(* Logix 5000 project; controller AMANA_DC_PLANT_01 vendor 1 type 14 code 164 rev 31.12; software revision 31.02; part 4 of 9 *)
(* tags used below, declared in another part *)
   Break_1stStation : BOOL;
   Break_LineWide : BOOL;
   Break_WorkCenter : BOOL;
   Break_Workstation : BOOL;
   Local_Timer : TIMER[10];
   LN00_1st_Station_Break_Code : DINT;
   LN00_FPY : REAL;
   LN00_MLC_Downtime : BOOL;
   LN00_Schedule : UDT_Current_Status;
   LN00_SNModel_MSG : MESSAGE;
   LN00_to_DC1_Main_Messages_0 : DINT[40];
   LN00_to_DC1_Main_Messages_1 : DINT[120];
   LN00_to_DC1_Main_Messages_2 : DINT[120];
   LN00_to_DC1_Main_Messages_3 : DINT[120];
   LN00_to_DC1_Main_Messages_4 : DINT[120];
   LN00_to_DC1_Main_Messages_5 : DINT[120];
   LN00_to_DC1_Main_MSG1 : MESSAGE;
   LN00_to_DC1_Main_MSG2 : MESSAGE;
   LN00_to_DC1_Main_MSG3 : MESSAGE;
   LN00_to_DC1_Main_MSG4 : MESSAGE;
   LN00_to_DC1_Main_MSG5 : MESSAGE;
   LN00_to_DC1_Main_MSG6 : MESSAGE;
   LN00DAM01 : DINT;
   LN00DAM02 : DINT;
   LN00DAM03 : DINT;
   LN00DAM04 : DINT;
   LN00DAM05 : DINT;
   LN00DAM06 : DINT;
   LN00DAM07 : DINT;
   LN00DAM08 : DINT;
   LN00DAM09 : DINT;
   LN00DBM02 : DINT;
   LN00DBM03 : DINT;
   LN00DCM04 : DINT;
   LN00DCM05 : DINT;
   LN00DCM06 : DINT;
   LN00DCM07 : DINT;
   LN00DCM08 : DINT;
   LN00DCM09 : DINT;
   LN00DCM10 : DINT;
   LN00DCM11 : DINT;
   LN00DCM12 : DINT;
   LN00DCM13 : DINT;
   LN00DCM14 : DINT;
   LN00DCM15 : DINT;
   LN00DCM16 : DINT;
   LN00DCM17 : DINT;
   LN00DCM18 : DINT;
   LN00DCM19 : DINT;
   LN00DCM20 : DINT;
   LN00DCM21 : DINT;
   LN00DCM22 : DINT;
   LN00DCM23 : DINT;
   LN00DCM24 : DINT;
   LN00DCM25 : DINT;
   LN00DCM26 : DINT;
   LN00DCM27 : DINT;
   LN00DCM28 : DINT;
   LN00DCM29 : DINT;
   LN00DCM30 : DINT;
   LN00DCM31 : DINT;
   LN00DCM32 : DINT;
   LN00DCM33 : DINT;
   LN00DCM34 : DINT;
   LN00DCM35 : DINT;
   LN00DCM36 : DINT;
   LN00DCM37 : DINT;
   LN00DCM38 : DINT;
   LN00DCM39 : DINT;
   LN00DCM40 : DINT;
   LN00DDM01 : DINT;
   LN00DDM02 : DINT;
   LN00DDM03 : DINT;
   LN00DDM04 : DINT;
   LN00DDM05 : DINT;
   LN00DDM06 : DINT;
   LN00DDM07 : DINT;
   LN00DDM08 : DINT;
   LN00DDM09 : DINT;
   LN00DDM10 : DINT;
   LN00DDM11 : DINT;
   LN00DDM12 : DINT;
   LN00DDM13 : DINT;
   LN00DDM14 : DINT;
   LN00DDM15 : DINT;
   LN00DDM16 : DINT;
   LN00DDM17 : DINT;
   LN00DDM18 : DINT;
   LN00DDM19 : DINT;
   LN00DDM20 : DINT;
   LN00DDM21 : DINT;
   LN00DDM22 : DINT;
   LN00DDM23 : DINT;
   LN00DDM24 : DINT;
   LN00DDM25 : DINT;
   LN00DDM26 : DINT;
   LN00DDM27 : DINT;
   LN00DDM28 : DINT;
   LN00DEM01 : DINT;
   LN00DEM02 : DINT;
   LN00DEM03 : DINT;
   LN00DEM04 : DINT;
   LN00DEM05 : DINT;
   LN00EAM00 : DINT;
   LN00EBM00 : DINT;
   LN00EDM00 : DINT;
(* LN00, continued *)

ROUTINE R03_DataFromLines   (* ladder *)
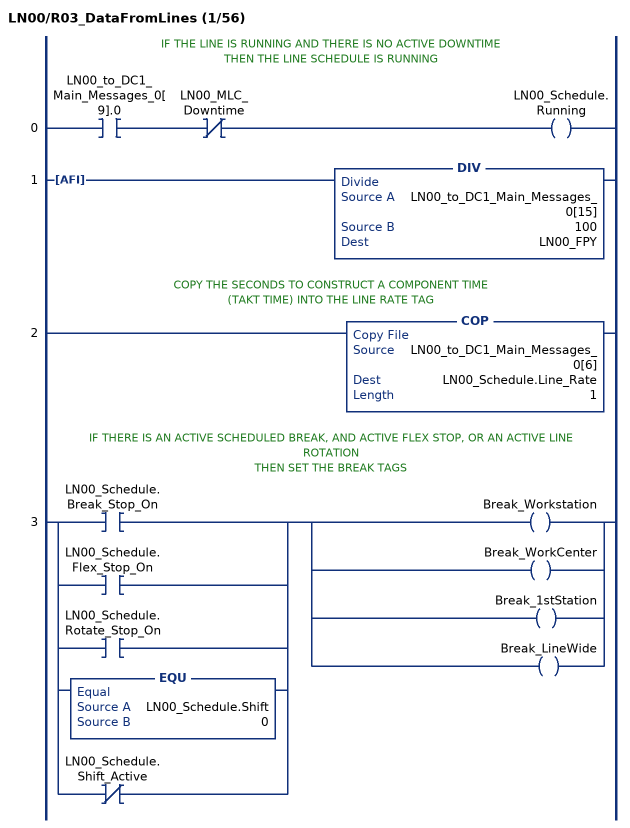
   // IF THE LINE IS RUNNING AND THERE IS NO ACTIVE DOWNTIME
   // THEN THE LINE SCHEDULE IS RUNNING
   0: XIC(LN00_to_DC1_Main_Messages_0[9].0)XIO(LN00_MLC_Downtime)OTE(LN00_Schedule.Running);
   1: AFI()DIV(LN00_to_DC1_Main_Messages_0[15],100,LN00_FPY);
   // COPY THE SECONDS TO CONSTRUCT A COMPONENT TIME
   // (TAKT TIME) INTO THE LINE RATE TAG
   2: COP(LN00_to_DC1_Main_Messages_0[6],LN00_Schedule.Line_Rate,1);
   // IF THERE IS AN ACTIVE SCHEDULED BREAK, AND ACTIVE FLEX STOP, OR AN ACTIVE LINE ROTATION
   // THEN SET THE BREAK TAGS
   3: [XIC(LN00_Schedule.Break_Stop_On) ,XIC(LN00_Schedule.Flex_Stop_On) ,XIC(LN00_Schedule.Rotate_Stop_On) ,EQU(LN00_Schedule.Shift,0) ,XIO(LN00_Schedule.Shift_Active) ][OTE(Break_Workstation) ,OTE(Break_WorkCenter) ,OTE(Break_1stStation) ,OTE(Break_LineWide) ];
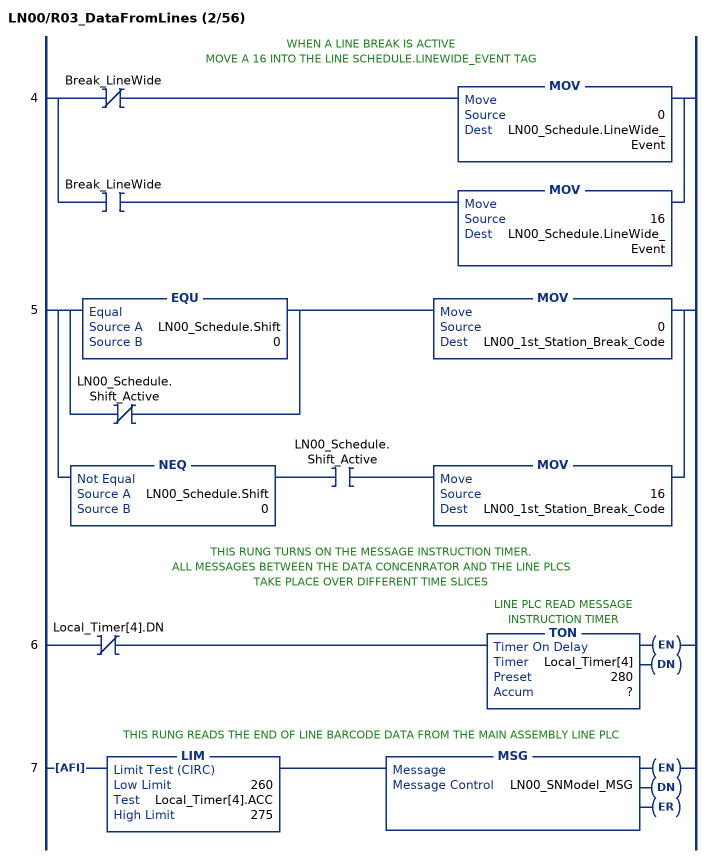
   // WHEN A LINE BREAK IS ACTIVE
   // MOVE A 16 INTO THE LINE SCHEDULE.LINEWIDE_EVENT TAG
   4: [XIO(Break_LineWide) MOV(0,LN00_Schedule.LineWide_Event) ,XIC(Break_LineWide) MOV(16,LN00_Schedule.LineWide_Event) ];
   5: [[EQU(LN00_Schedule.Shift,0) ,XIO(LN00_Schedule.Shift_Active) ] MOV(0,LN00_1st_Station_Break_Code) ,NEQ(LN00_Schedule.Shift,0) XIC(LN00_Schedule.Shift_Active) MOV(16,LN00_1st_Station_Break_Code) ];
   // THIS RUNG TURNS ON THE MESSAGE INSTRUCTION TIMER.
   // ALL MESSAGES BETWEEN THE DATA CONCENRATOR AND THE LINE PLCS
   // TAKE PLACE OVER DIFFERENT TIME SLICES
   6: XIO(Local_Timer[4].DN)TON(Local_Timer[4],?,?);
   // THIS RUNG READS THE END OF LINE BARCODE DATA FROM THE MAIN ASSEMBLY LINE PLC
   7: AFI()LIM(260,Local_Timer[4].ACC,275)MSG(LN00_SNModel_MSG);
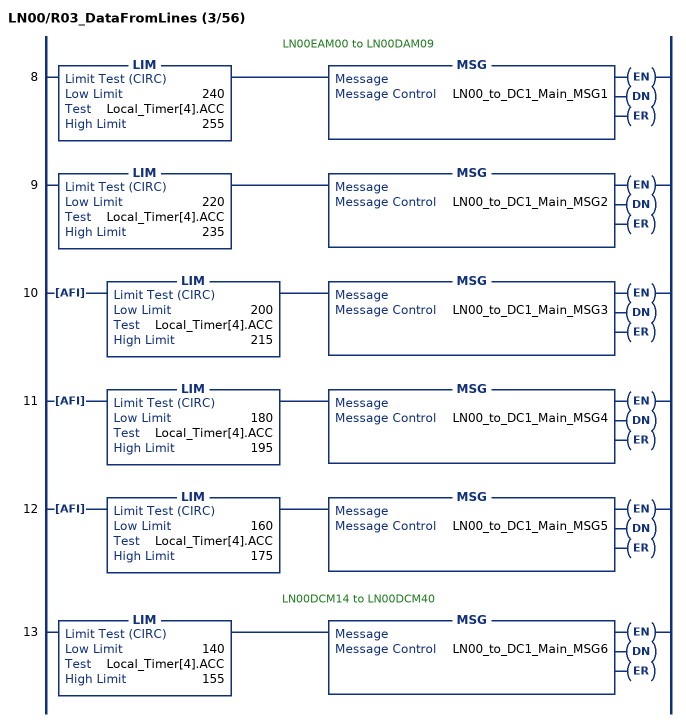
   // LN00EAM00 to LN00DAM09
   8: LIM(240,Local_Timer[4].ACC,255)MSG(LN00_to_DC1_Main_MSG1);
   9: LIM(220,Local_Timer[4].ACC,235)MSG(LN00_to_DC1_Main_MSG2);
   10: AFI()LIM(200,Local_Timer[4].ACC,215)MSG(LN00_to_DC1_Main_MSG3);
   11: AFI()LIM(180,Local_Timer[4].ACC,195)MSG(LN00_to_DC1_Main_MSG4);
   12: AFI()LIM(160,Local_Timer[4].ACC,175)MSG(LN00_to_DC1_Main_MSG5);
   // LN00DCM14 to LN00DCM40
   13: LIM(140,Local_Timer[4].ACC,155)MSG(LN00_to_DC1_Main_MSG6);
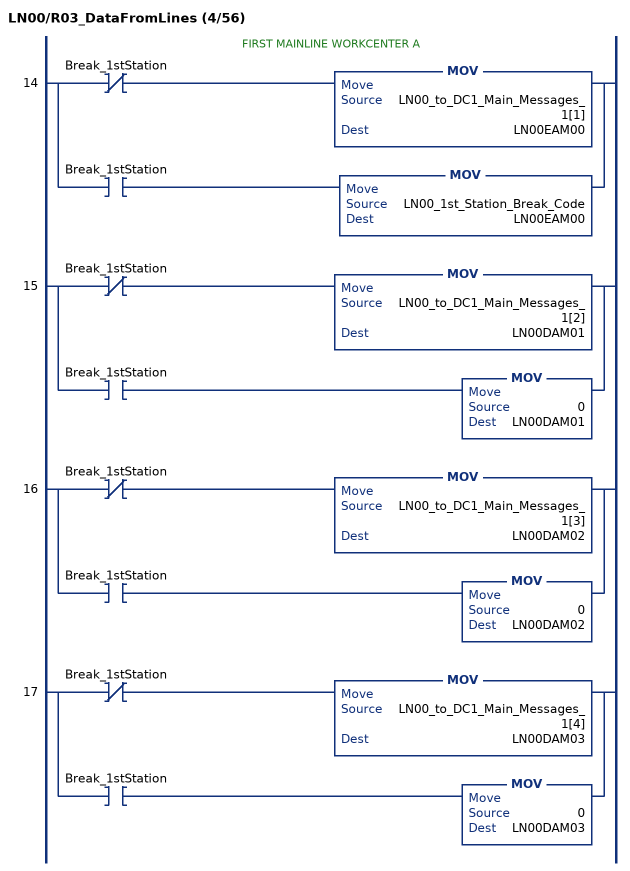
   // FIRST MAINLINE WORKCENTER A
   14: [XIO(Break_1stStation) MOV(LN00_to_DC1_Main_Messages_1[1],LN00EAM00) ,XIC(Break_1stStation) MOV(LN00_1st_Station_Break_Code,LN00EAM00) ];
   15: [XIO(Break_1stStation) MOV(LN00_to_DC1_Main_Messages_1[2],LN00DAM01) ,XIC(Break_1stStation) MOV(0,LN00DAM01) ];
   16: [XIO(Break_1stStation) MOV(LN00_to_DC1_Main_Messages_1[3],LN00DAM02) ,XIC(Break_1stStation) MOV(0,LN00DAM02) ];
   17: [XIO(Break_1stStation) MOV(LN00_to_DC1_Main_Messages_1[4],LN00DAM03) ,XIC(Break_1stStation) MOV(0,LN00DAM03) ];
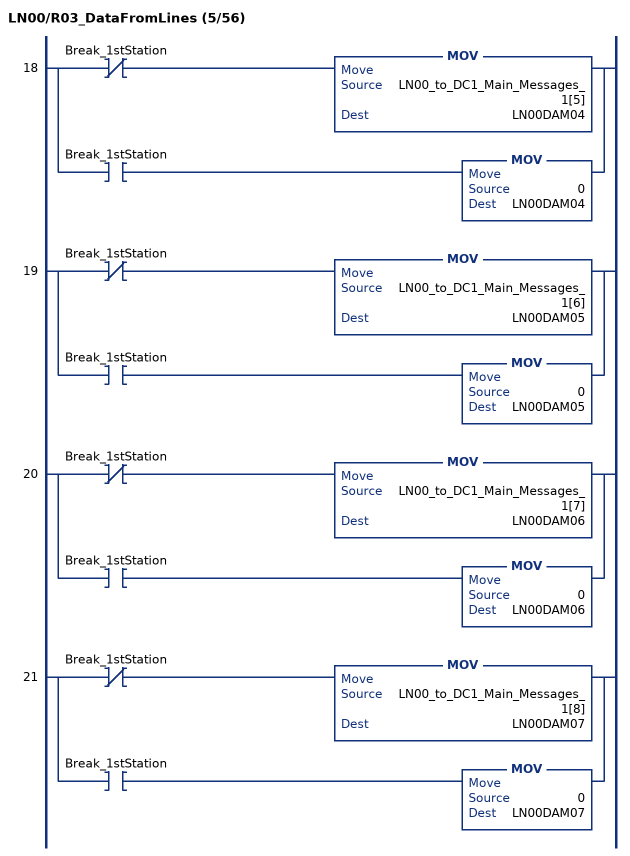
   18: [XIO(Break_1stStation) MOV(LN00_to_DC1_Main_Messages_1[5],LN00DAM04) ,XIC(Break_1stStation) MOV(0,LN00DAM04) ];
   19: [XIO(Break_1stStation) MOV(LN00_to_DC1_Main_Messages_1[6],LN00DAM05) ,XIC(Break_1stStation) MOV(0,LN00DAM05) ];
   20: [XIO(Break_1stStation) MOV(LN00_to_DC1_Main_Messages_1[7],LN00DAM06) ,XIC(Break_1stStation) MOV(0,LN00DAM06) ];
   21: [XIO(Break_1stStation) MOV(LN00_to_DC1_Main_Messages_1[8],LN00DAM07) ,XIC(Break_1stStation) MOV(0,LN00DAM07) ];
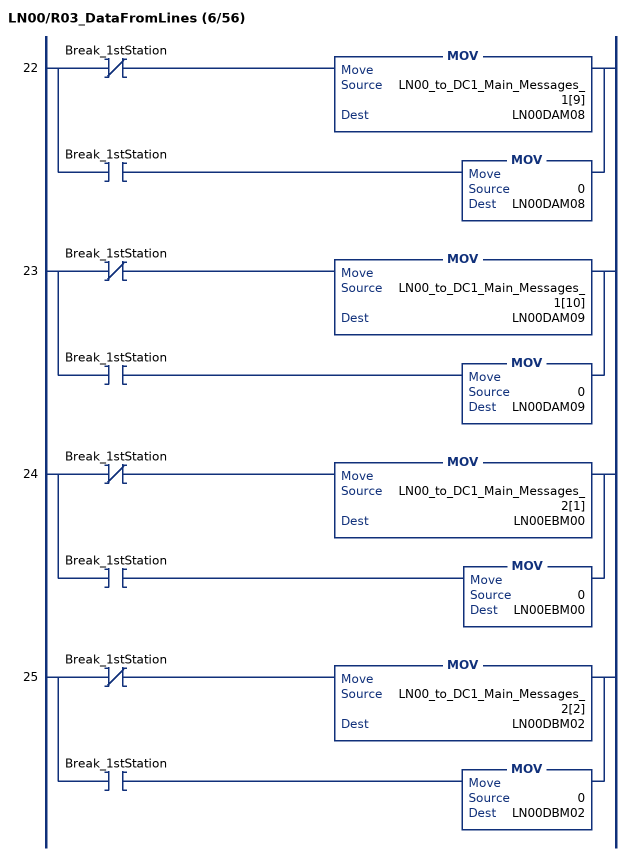
   22: [XIO(Break_1stStation) MOV(LN00_to_DC1_Main_Messages_1[9],LN00DAM08) ,XIC(Break_1stStation) MOV(0,LN00DAM08) ];
   23: [XIO(Break_1stStation) MOV(LN00_to_DC1_Main_Messages_1[10],LN00DAM09) ,XIC(Break_1stStation) MOV(0,LN00DAM09) ];
   24: [XIO(Break_1stStation) MOV(LN00_to_DC1_Main_Messages_2[1],LN00EBM00) ,XIC(Break_1stStation) MOV(0,LN00EBM00) ];
   25: [XIO(Break_1stStation) MOV(LN00_to_DC1_Main_Messages_2[2],LN00DBM02) ,XIC(Break_1stStation) MOV(0,LN00DBM02) ];
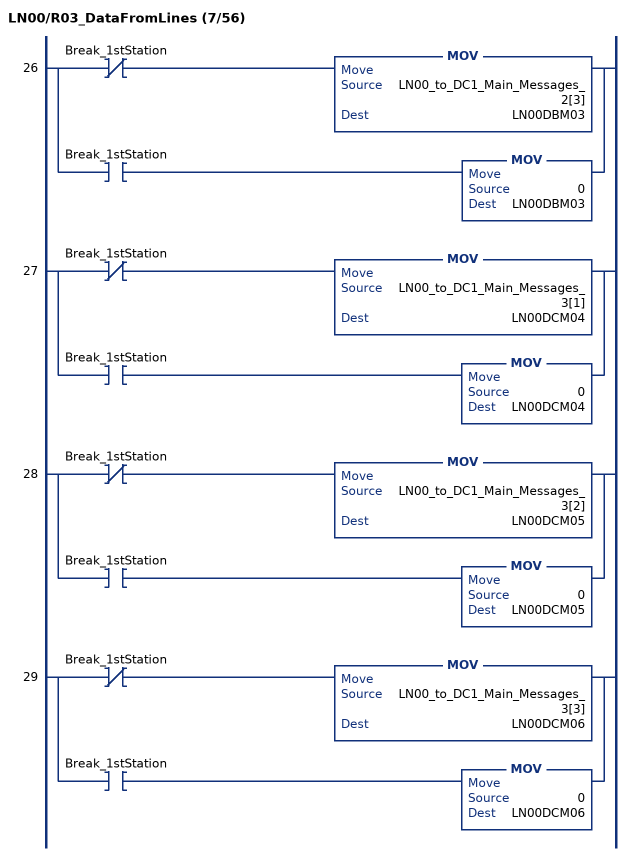
   26: [XIO(Break_1stStation) MOV(LN00_to_DC1_Main_Messages_2[3],LN00DBM03) ,XIC(Break_1stStation) MOV(0,LN00DBM03) ];
   27: [XIO(Break_1stStation) MOV(LN00_to_DC1_Main_Messages_3[1],LN00DCM04) ,XIC(Break_1stStation) MOV(0,LN00DCM04) ];
   28: [XIO(Break_1stStation) MOV(LN00_to_DC1_Main_Messages_3[2],LN00DCM05) ,XIC(Break_1stStation) MOV(0,LN00DCM05) ];
   29: [XIO(Break_1stStation) MOV(LN00_to_DC1_Main_Messages_3[3],LN00DCM06) ,XIC(Break_1stStation) MOV(0,LN00DCM06) ];
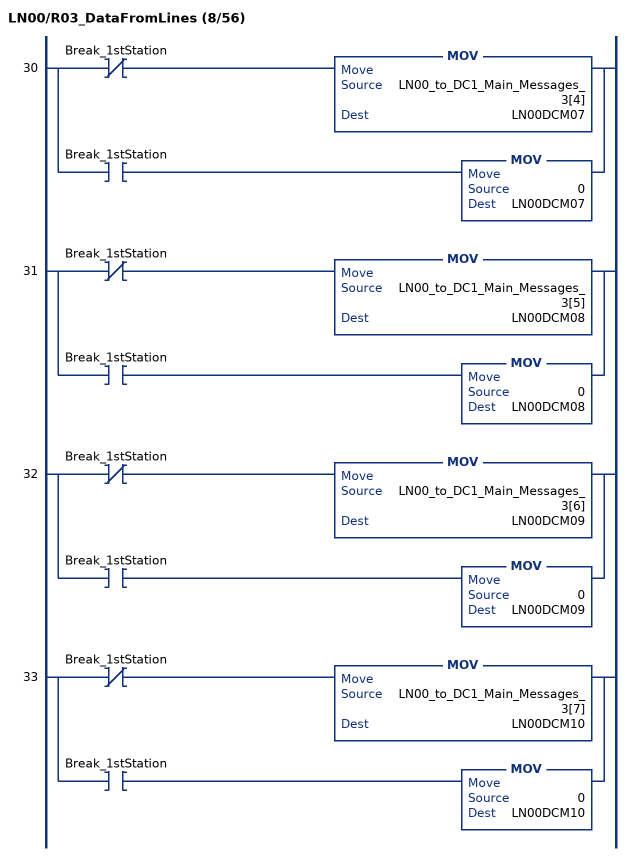
   30: [XIO(Break_1stStation) MOV(LN00_to_DC1_Main_Messages_3[4],LN00DCM07) ,XIC(Break_1stStation) MOV(0,LN00DCM07) ];
   31: [XIO(Break_1stStation) MOV(LN00_to_DC1_Main_Messages_3[5],LN00DCM08) ,XIC(Break_1stStation) MOV(0,LN00DCM08) ];
   32: [XIO(Break_1stStation) MOV(LN00_to_DC1_Main_Messages_3[6],LN00DCM09) ,XIC(Break_1stStation) MOV(0,LN00DCM09) ];
   33: [XIO(Break_1stStation) MOV(LN00_to_DC1_Main_Messages_3[7],LN00DCM10) ,XIC(Break_1stStation) MOV(0,LN00DCM10) ];
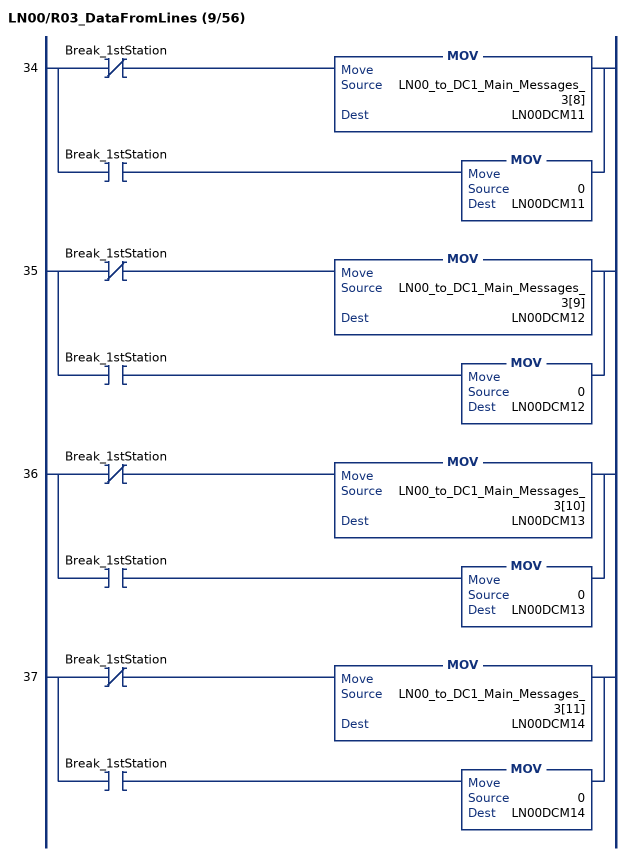
   34: [XIO(Break_1stStation) MOV(LN00_to_DC1_Main_Messages_3[8],LN00DCM11) ,XIC(Break_1stStation) MOV(0,LN00DCM11) ];
   35: [XIO(Break_1stStation) MOV(LN00_to_DC1_Main_Messages_3[9],LN00DCM12) ,XIC(Break_1stStation) MOV(0,LN00DCM12) ];
   36: [XIO(Break_1stStation) MOV(LN00_to_DC1_Main_Messages_3[10],LN00DCM13) ,XIC(Break_1stStation) MOV(0,LN00DCM13) ];
   37: [XIO(Break_1stStation) MOV(LN00_to_DC1_Main_Messages_3[11],LN00DCM14) ,XIC(Break_1stStation) MOV(0,LN00DCM14) ];
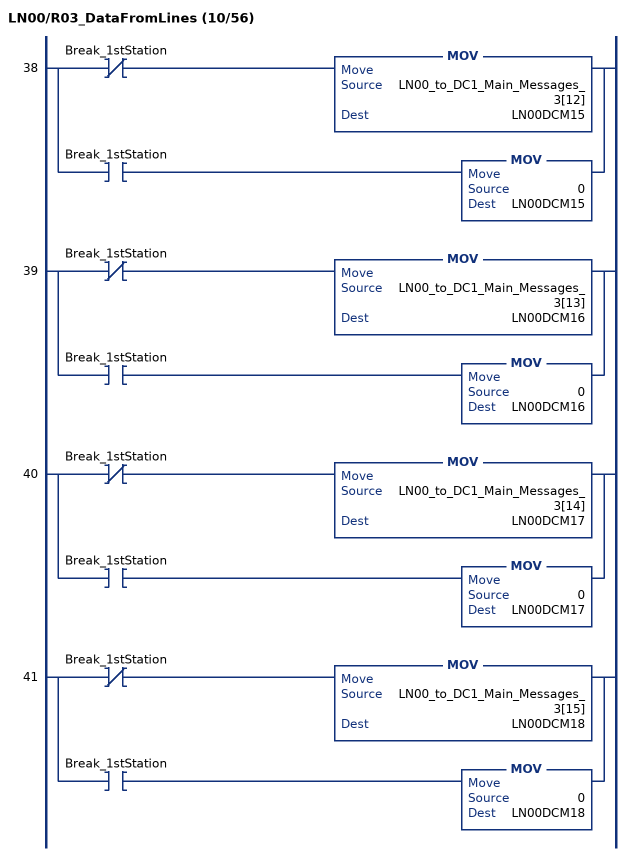
   38: [XIO(Break_1stStation) MOV(LN00_to_DC1_Main_Messages_3[12],LN00DCM15) ,XIC(Break_1stStation) MOV(0,LN00DCM15) ];
   39: [XIO(Break_1stStation) MOV(LN00_to_DC1_Main_Messages_3[13],LN00DCM16) ,XIC(Break_1stStation) MOV(0,LN00DCM16) ];
   40: [XIO(Break_1stStation) MOV(LN00_to_DC1_Main_Messages_3[14],LN00DCM17) ,XIC(Break_1stStation) MOV(0,LN00DCM17) ];
   41: [XIO(Break_1stStation) MOV(LN00_to_DC1_Main_Messages_3[15],LN00DCM18) ,XIC(Break_1stStation) MOV(0,LN00DCM18) ];
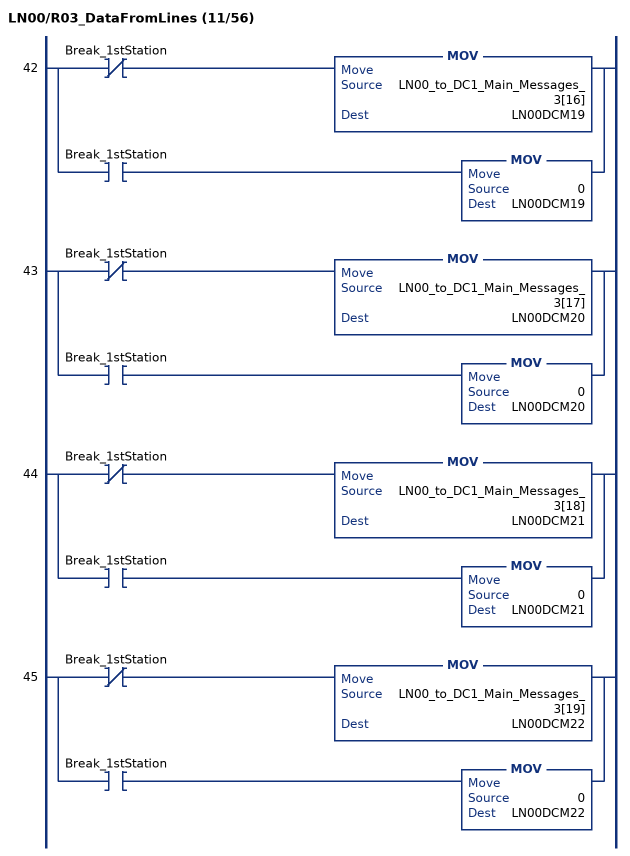
   42: [XIO(Break_1stStation) MOV(LN00_to_DC1_Main_Messages_3[16],LN00DCM19) ,XIC(Break_1stStation) MOV(0,LN00DCM19) ];
   43: [XIO(Break_1stStation) MOV(LN00_to_DC1_Main_Messages_3[17],LN00DCM20) ,XIC(Break_1stStation) MOV(0,LN00DCM20) ];
   44: [XIO(Break_1stStation) MOV(LN00_to_DC1_Main_Messages_3[18],LN00DCM21) ,XIC(Break_1stStation) MOV(0,LN00DCM21) ];
   45: [XIO(Break_1stStation) MOV(LN00_to_DC1_Main_Messages_3[19],LN00DCM22) ,XIC(Break_1stStation) MOV(0,LN00DCM22) ];
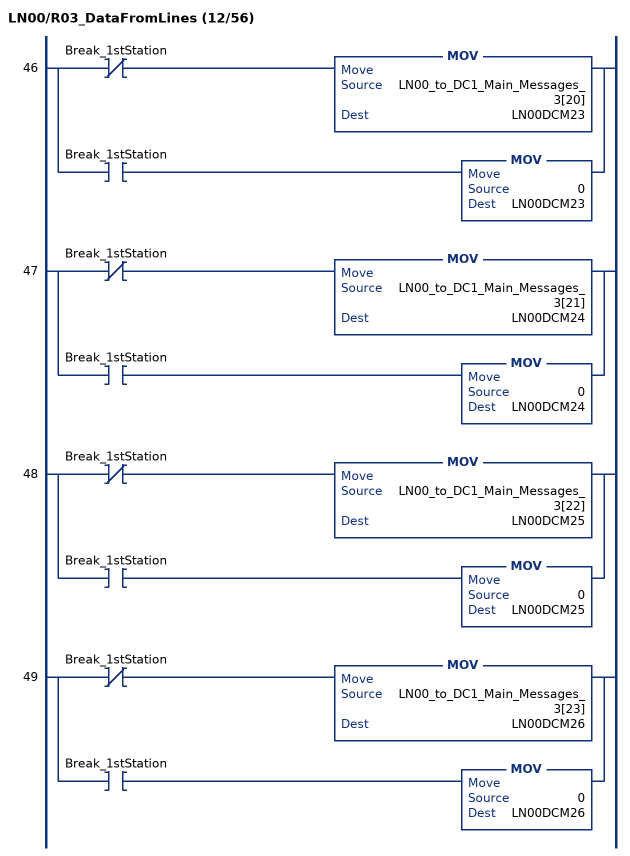
   46: [XIO(Break_1stStation) MOV(LN00_to_DC1_Main_Messages_3[20],LN00DCM23) ,XIC(Break_1stStation) MOV(0,LN00DCM23) ];
   47: [XIO(Break_1stStation) MOV(LN00_to_DC1_Main_Messages_3[21],LN00DCM24) ,XIC(Break_1stStation) MOV(0,LN00DCM24) ];
   48: [XIO(Break_1stStation) MOV(LN00_to_DC1_Main_Messages_3[22],LN00DCM25) ,XIC(Break_1stStation) MOV(0,LN00DCM25) ];
   49: [XIO(Break_1stStation) MOV(LN00_to_DC1_Main_Messages_3[23],LN00DCM26) ,XIC(Break_1stStation) MOV(0,LN00DCM26) ];
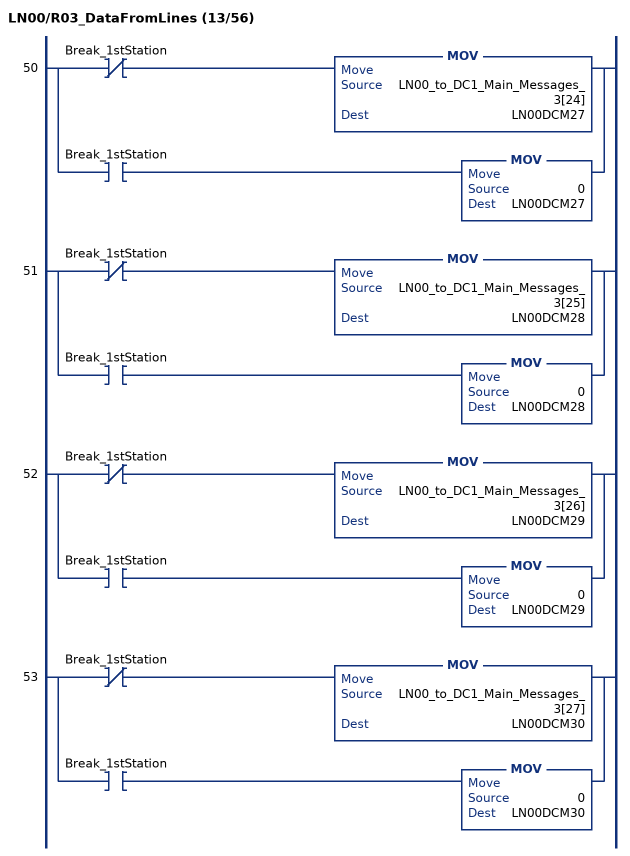
   50: [XIO(Break_1stStation) MOV(LN00_to_DC1_Main_Messages_3[24],LN00DCM27) ,XIC(Break_1stStation) MOV(0,LN00DCM27) ];
   51: [XIO(Break_1stStation) MOV(LN00_to_DC1_Main_Messages_3[25],LN00DCM28) ,XIC(Break_1stStation) MOV(0,LN00DCM28) ];
   52: [XIO(Break_1stStation) MOV(LN00_to_DC1_Main_Messages_3[26],LN00DCM29) ,XIC(Break_1stStation) MOV(0,LN00DCM29) ];
   53: [XIO(Break_1stStation) MOV(LN00_to_DC1_Main_Messages_3[27],LN00DCM30) ,XIC(Break_1stStation) MOV(0,LN00DCM30) ];
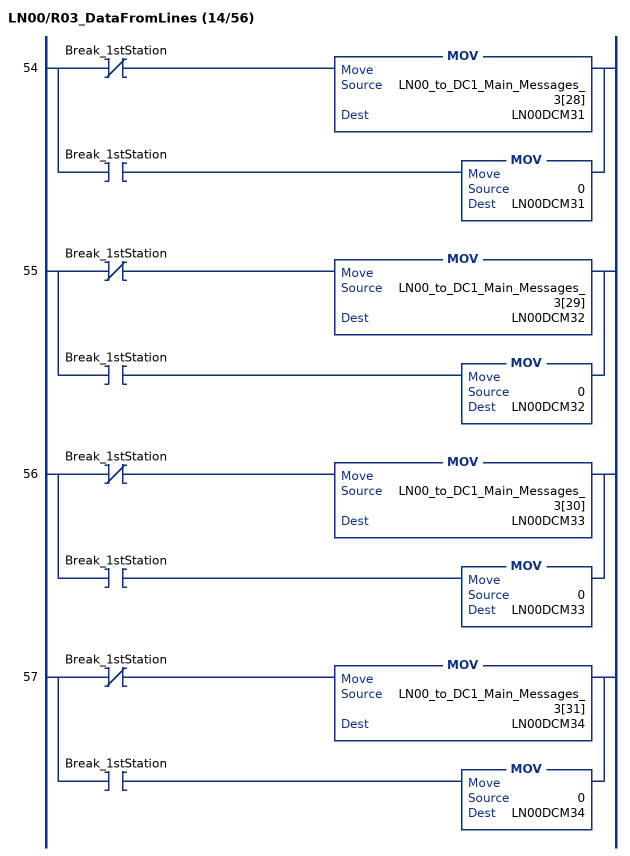
   54: [XIO(Break_1stStation) MOV(LN00_to_DC1_Main_Messages_3[28],LN00DCM31) ,XIC(Break_1stStation) MOV(0,LN00DCM31) ];
   55: [XIO(Break_1stStation) MOV(LN00_to_DC1_Main_Messages_3[29],LN00DCM32) ,XIC(Break_1stStation) MOV(0,LN00DCM32) ];
   56: [XIO(Break_1stStation) MOV(LN00_to_DC1_Main_Messages_3[30],LN00DCM33) ,XIC(Break_1stStation) MOV(0,LN00DCM33) ];
   57: [XIO(Break_1stStation) MOV(LN00_to_DC1_Main_Messages_3[31],LN00DCM34) ,XIC(Break_1stStation) MOV(0,LN00DCM34) ];
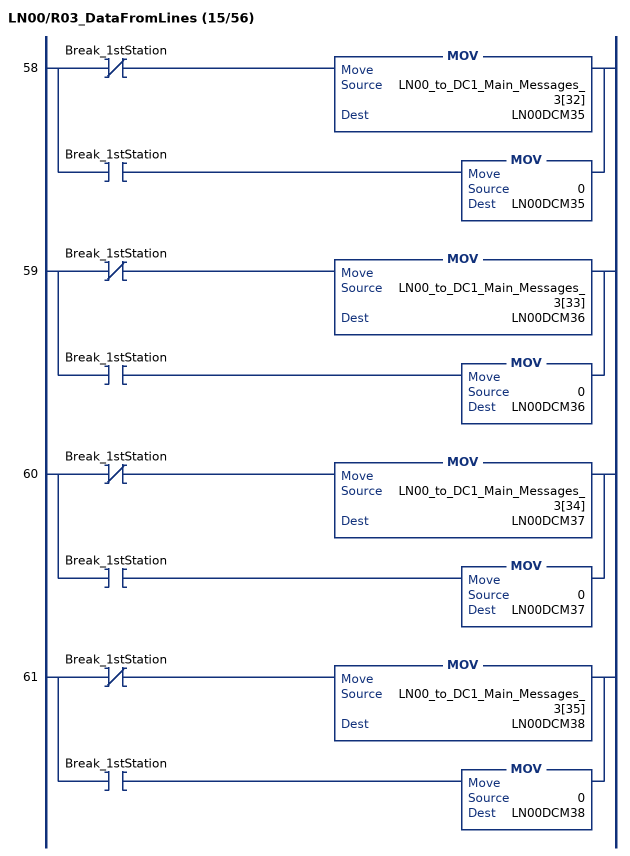
   58: [XIO(Break_1stStation) MOV(LN00_to_DC1_Main_Messages_3[32],LN00DCM35) ,XIC(Break_1stStation) MOV(0,LN00DCM35) ];
   59: [XIO(Break_1stStation) MOV(LN00_to_DC1_Main_Messages_3[33],LN00DCM36) ,XIC(Break_1stStation) MOV(0,LN00DCM36) ];
   60: [XIO(Break_1stStation) MOV(LN00_to_DC1_Main_Messages_3[34],LN00DCM37) ,XIC(Break_1stStation) MOV(0,LN00DCM37) ];
   61: [XIO(Break_1stStation) MOV(LN00_to_DC1_Main_Messages_3[35],LN00DCM38) ,XIC(Break_1stStation) MOV(0,LN00DCM38) ];
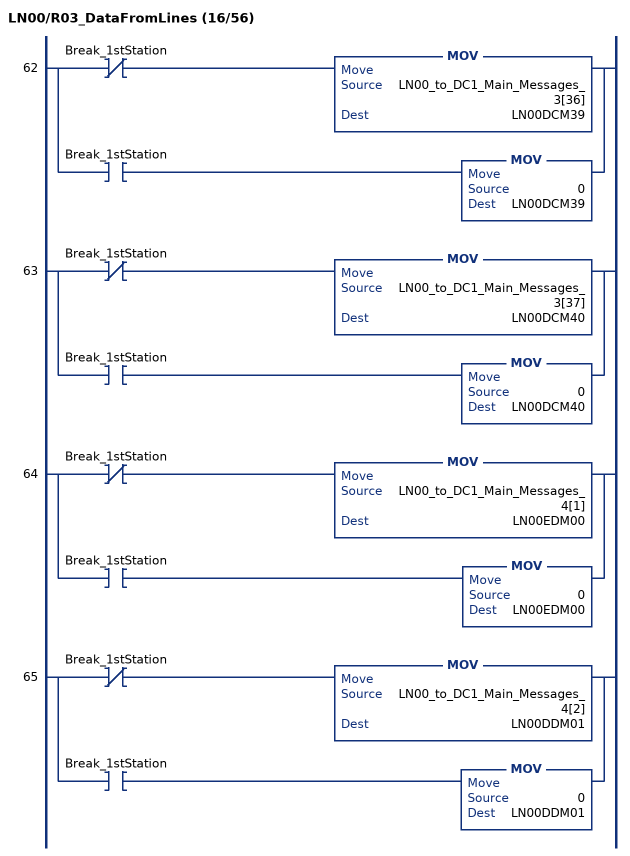
   62: [XIO(Break_1stStation) MOV(LN00_to_DC1_Main_Messages_3[36],LN00DCM39) ,XIC(Break_1stStation) MOV(0,LN00DCM39) ];
   63: [XIO(Break_1stStation) MOV(LN00_to_DC1_Main_Messages_3[37],LN00DCM40) ,XIC(Break_1stStation) MOV(0,LN00DCM40) ];
   64: [XIO(Break_1stStation) MOV(LN00_to_DC1_Main_Messages_4[1],LN00EDM00) ,XIC(Break_1stStation) MOV(0,LN00EDM00) ];
   65: [XIO(Break_1stStation) MOV(LN00_to_DC1_Main_Messages_4[2],LN00DDM01) ,XIC(Break_1stStation) MOV(0,LN00DDM01) ];
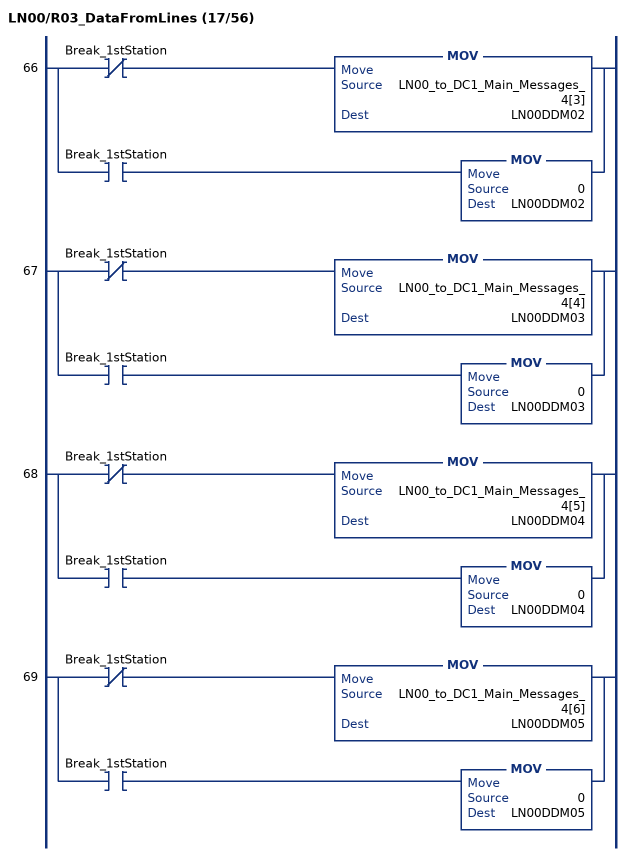
   66: [XIO(Break_1stStation) MOV(LN00_to_DC1_Main_Messages_4[3],LN00DDM02) ,XIC(Break_1stStation) MOV(0,LN00DDM02) ];
   67: [XIO(Break_1stStation) MOV(LN00_to_DC1_Main_Messages_4[4],LN00DDM03) ,XIC(Break_1stStation) MOV(0,LN00DDM03) ];
   68: [XIO(Break_1stStation) MOV(LN00_to_DC1_Main_Messages_4[5],LN00DDM04) ,XIC(Break_1stStation) MOV(0,LN00DDM04) ];
   69: [XIO(Break_1stStation) MOV(LN00_to_DC1_Main_Messages_4[6],LN00DDM05) ,XIC(Break_1stStation) MOV(0,LN00DDM05) ];
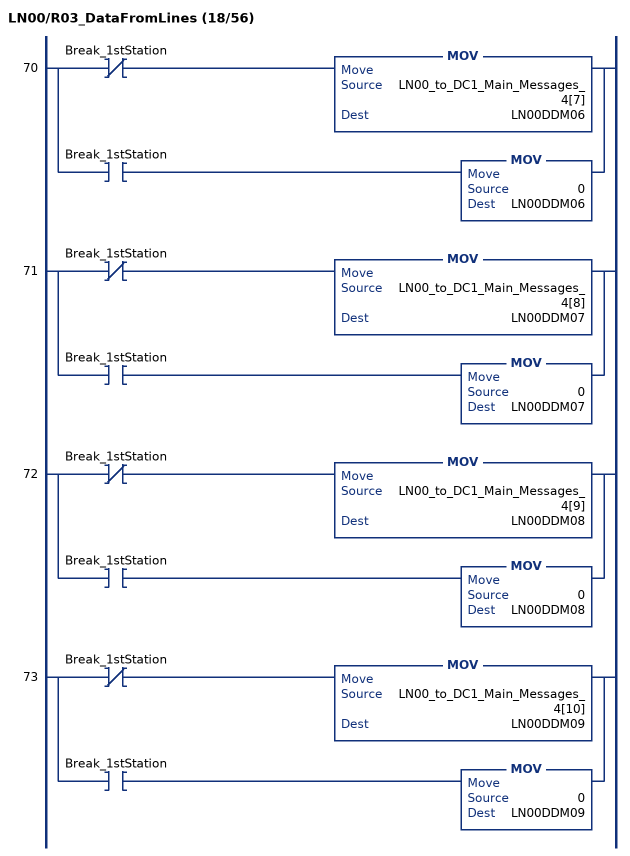
   70: [XIO(Break_1stStation) MOV(LN00_to_DC1_Main_Messages_4[7],LN00DDM06) ,XIC(Break_1stStation) MOV(0,LN00DDM06) ];
   71: [XIO(Break_1stStation) MOV(LN00_to_DC1_Main_Messages_4[8],LN00DDM07) ,XIC(Break_1stStation) MOV(0,LN00DDM07) ];
   72: [XIO(Break_1stStation) MOV(LN00_to_DC1_Main_Messages_4[9],LN00DDM08) ,XIC(Break_1stStation) MOV(0,LN00DDM08) ];
   73: [XIO(Break_1stStation) MOV(LN00_to_DC1_Main_Messages_4[10],LN00DDM09) ,XIC(Break_1stStation) MOV(0,LN00DDM09) ];
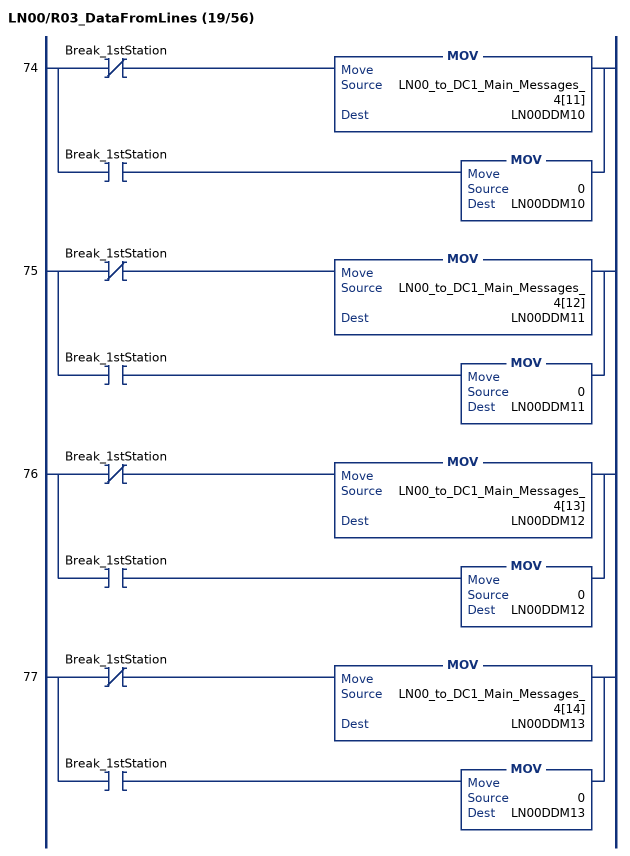
   74: [XIO(Break_1stStation) MOV(LN00_to_DC1_Main_Messages_4[11],LN00DDM10) ,XIC(Break_1stStation) MOV(0,LN00DDM10) ];
   75: [XIO(Break_1stStation) MOV(LN00_to_DC1_Main_Messages_4[12],LN00DDM11) ,XIC(Break_1stStation) MOV(0,LN00DDM11) ];
   76: [XIO(Break_1stStation) MOV(LN00_to_DC1_Main_Messages_4[13],LN00DDM12) ,XIC(Break_1stStation) MOV(0,LN00DDM12) ];
   77: [XIO(Break_1stStation) MOV(LN00_to_DC1_Main_Messages_4[14],LN00DDM13) ,XIC(Break_1stStation) MOV(0,LN00DDM13) ];
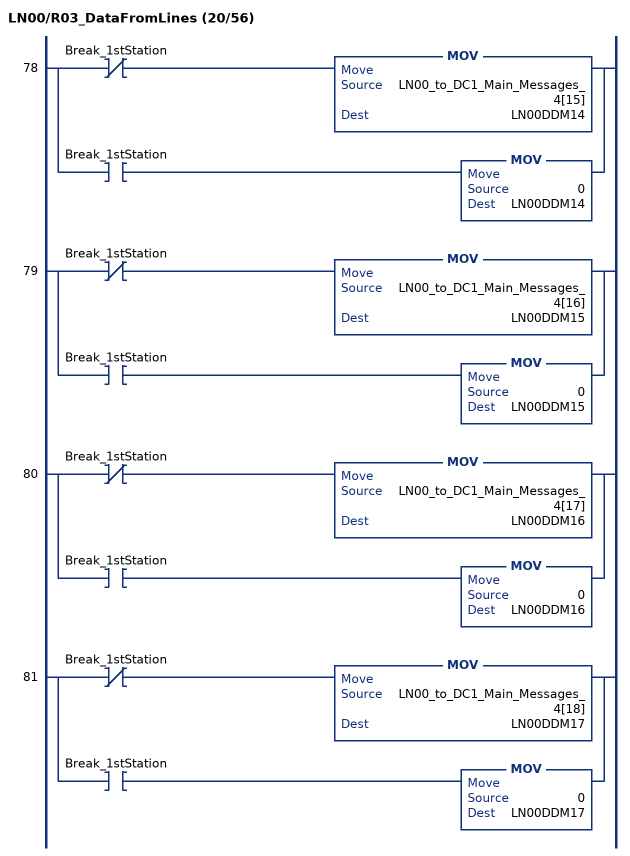
   78: [XIO(Break_1stStation) MOV(LN00_to_DC1_Main_Messages_4[15],LN00DDM14) ,XIC(Break_1stStation) MOV(0,LN00DDM14) ];
   79: [XIO(Break_1stStation) MOV(LN00_to_DC1_Main_Messages_4[16],LN00DDM15) ,XIC(Break_1stStation) MOV(0,LN00DDM15) ];
   80: [XIO(Break_1stStation) MOV(LN00_to_DC1_Main_Messages_4[17],LN00DDM16) ,XIC(Break_1stStation) MOV(0,LN00DDM16) ];
   81: [XIO(Break_1stStation) MOV(LN00_to_DC1_Main_Messages_4[18],LN00DDM17) ,XIC(Break_1stStation) MOV(0,LN00DDM17) ];
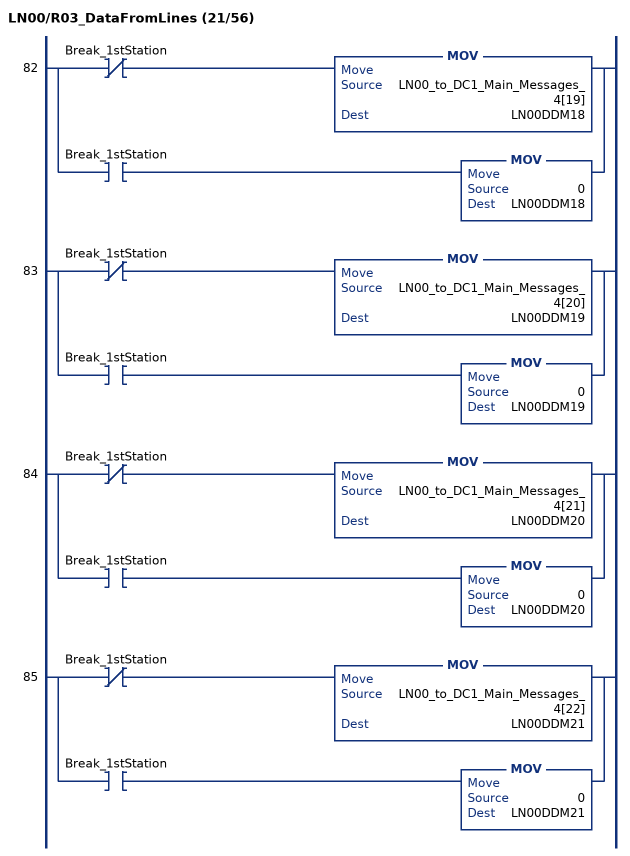
   82: [XIO(Break_1stStation) MOV(LN00_to_DC1_Main_Messages_4[19],LN00DDM18) ,XIC(Break_1stStation) MOV(0,LN00DDM18) ];
   83: [XIO(Break_1stStation) MOV(LN00_to_DC1_Main_Messages_4[20],LN00DDM19) ,XIC(Break_1stStation) MOV(0,LN00DDM19) ];
   84: [XIO(Break_1stStation) MOV(LN00_to_DC1_Main_Messages_4[21],LN00DDM20) ,XIC(Break_1stStation) MOV(0,LN00DDM20) ];
   85: [XIO(Break_1stStation) MOV(LN00_to_DC1_Main_Messages_4[22],LN00DDM21) ,XIC(Break_1stStation) MOV(0,LN00DDM21) ];
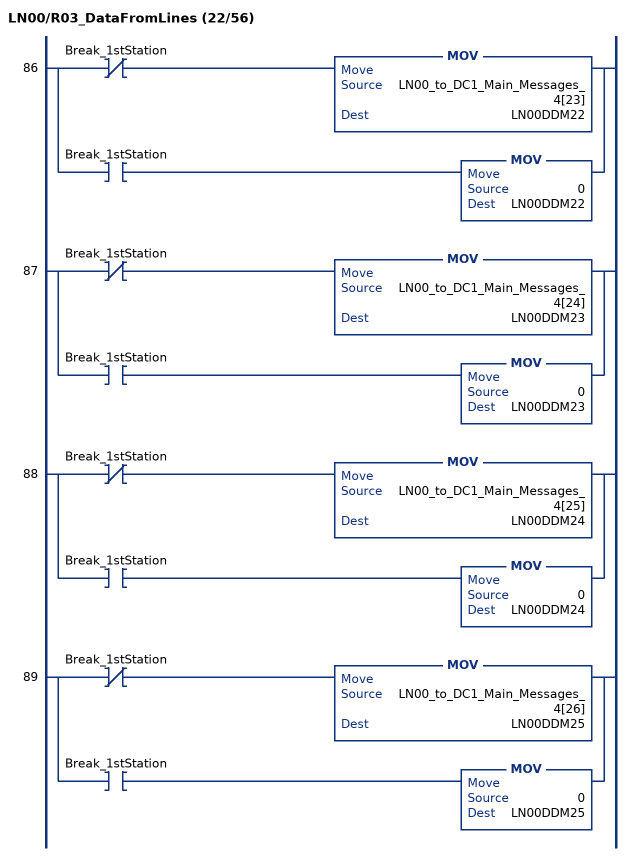
   86: [XIO(Break_1stStation) MOV(LN00_to_DC1_Main_Messages_4[23],LN00DDM22) ,XIC(Break_1stStation) MOV(0,LN00DDM22) ];
   87: [XIO(Break_1stStation) MOV(LN00_to_DC1_Main_Messages_4[24],LN00DDM23) ,XIC(Break_1stStation) MOV(0,LN00DDM23) ];
   88: [XIO(Break_1stStation) MOV(LN00_to_DC1_Main_Messages_4[25],LN00DDM24) ,XIC(Break_1stStation) MOV(0,LN00DDM24) ];
   89: [XIO(Break_1stStation) MOV(LN00_to_DC1_Main_Messages_4[26],LN00DDM25) ,XIC(Break_1stStation) MOV(0,LN00DDM25) ];
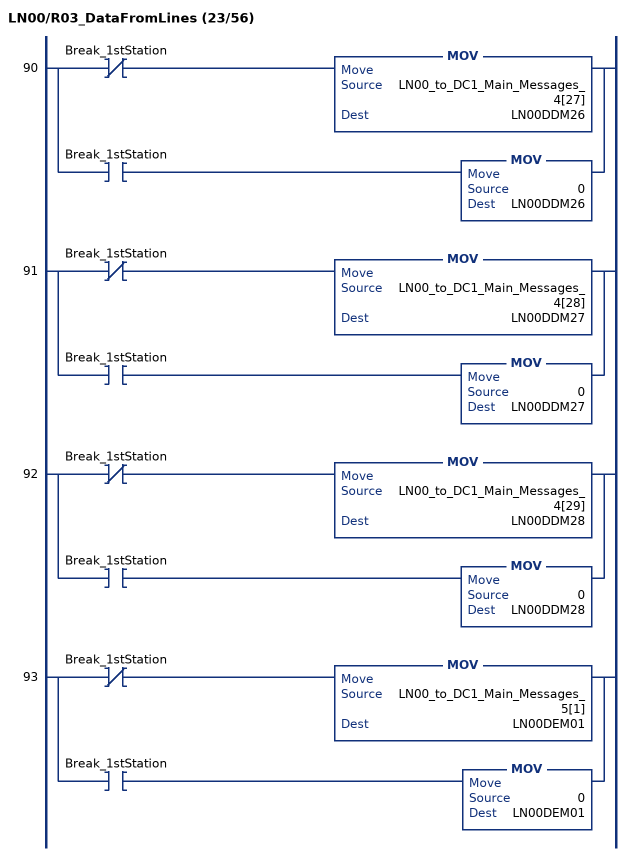
   90: [XIO(Break_1stStation) MOV(LN00_to_DC1_Main_Messages_4[27],LN00DDM26) ,XIC(Break_1stStation) MOV(0,LN00DDM26) ];
   91: [XIO(Break_1stStation) MOV(LN00_to_DC1_Main_Messages_4[28],LN00DDM27) ,XIC(Break_1stStation) MOV(0,LN00DDM27) ];
   92: [XIO(Break_1stStation) MOV(LN00_to_DC1_Main_Messages_4[29],LN00DDM28) ,XIC(Break_1stStation) MOV(0,LN00DDM28) ];
   93: [XIO(Break_1stStation) MOV(LN00_to_DC1_Main_Messages_5[1],LN00DEM01) ,XIC(Break_1stStation) MOV(0,LN00DEM01) ];
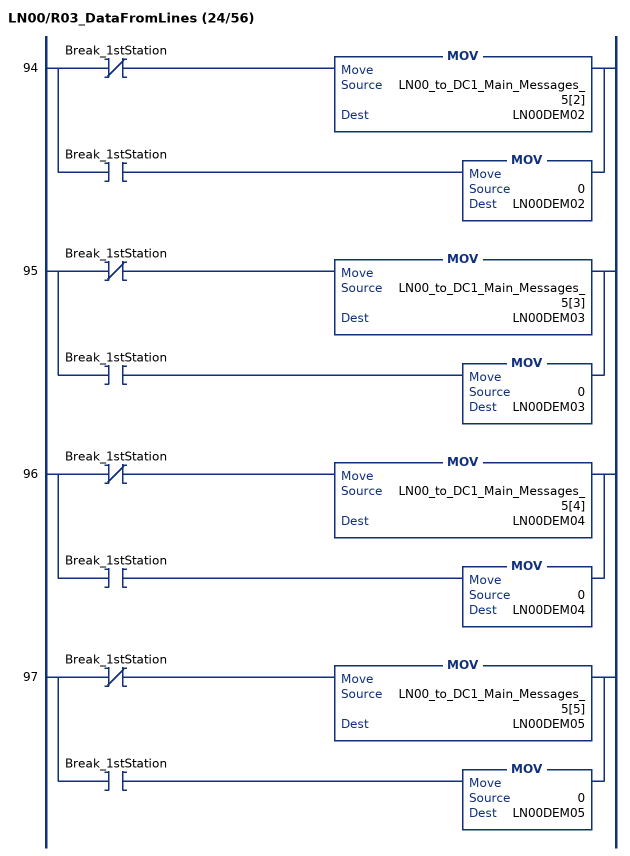
   94: [XIO(Break_1stStation) MOV(LN00_to_DC1_Main_Messages_5[2],LN00DEM02) ,XIC(Break_1stStation) MOV(0,LN00DEM02) ];
   95: [XIO(Break_1stStation) MOV(LN00_to_DC1_Main_Messages_5[3],LN00DEM03) ,XIC(Break_1stStation) MOV(0,LN00DEM03) ];
   96: [XIO(Break_1stStation) MOV(LN00_to_DC1_Main_Messages_5[4],LN00DEM04) ,XIC(Break_1stStation) MOV(0,LN00DEM04) ];
   97: [XIO(Break_1stStation) MOV(LN00_to_DC1_Main_Messages_5[5],LN00DEM05) ,XIC(Break_1stStation) MOV(0,LN00DEM05) ];
